{attribute addProperty BoxType "EL3632-0000-0022"}
{attribute addProperty Id "STATUSAT %I*STATUS_84521898162"}
{attribute addProperty CRC "3729672571"}
{attribute addProperty SizeInBites "16"}
{attribute addProperty SizeInBytes "2"}
TYPE Ch2_Status_DE4E497B :
STRUCT
	{attribute addProperty Name "STATUS"}
	STATUS AT %I* : STATUS_84521898;
END_STRUCT
END_TYPE

(* stored: Version 1.2.0.0, ProductVersion 3.1.4024.9
   DUT Ch2_Status_DE4E497B: Id {5699c7af-2671-45f2-ae8b-0f260b6611e1} *)
